// TIA Portal V17 export
// export: Created 2023-12-22T15:05:28.6996043Z, ExportSetting WithDefaults, DisplayName Totally Integrated Automation Portal, DisplayVersion V17, DisplayName TIA Portal Openness, DisplayVersion V17, DisplayName TIA Portal Version Control Interface, DisplayVersion V17, DisplayName STEP 7 Professional, DisplayVersion V17, DisplayName STEP 7 Safety, DisplayVersion V17, DisplayName WinCC Advanced, DisplayVersion V17
FUNCTION_BLOCK "Motors"   // FB240, LAD
{ S7_Optimized_Access := 'FALSE' }
VERSION : 0.1
// stored: AutoNumber false, IsIECCheckEnabled false, SetENOAutomatically false, UDAEnableTagReadback false
   VAR DB_SPECIFIC
      Time_DTL { S7_SetPoint := 'True'} : DTL;
   END_VAR
   VAR_TEMP   // added for the SCL form of the ladder/FBD networks
      _w1 : Bool;
   END_VAR
BEGIN

REGION Network 1: Электролизер / Мешалки
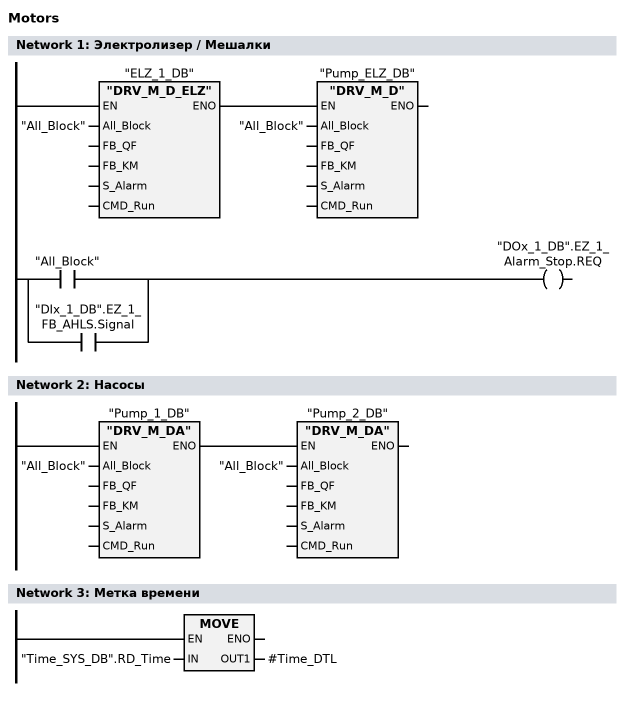
   RUNG wire#powerrail
      "ELZ_1_DB"(All_Block := "All_Block", FB_QF :=, FB_KM :=, S_Alarm :=, CMD_Run :=)
      "Pump_ELZ_DB"(All_Block := "All_Block", FB_QF :=, FB_KM :=, S_Alarm :=, CMD_Run :=)
   END_RUNG
   RUNG wire#powerrail
      Contact( "All_Block" )
      wire#w1
      Coil( "DOx_1_DB".EZ_1_Alarm_Stop.REQ )
   END_RUNG
   RUNG wire#powerrail
      Contact( "DIx_1_DB".EZ_1_FB_AHLS.Signal )
   END_RUNG wire#w1
   // the same network as SCL:
   "ELZ_1_DB"(All_Block := "All_Block", ENO => #_w1);   // "DRV_M_D_ELZ"
   IF #_w1 THEN
       "Pump_ELZ_DB"(All_Block := "All_Block");   // "DRV_M_D"
   END_IF;
   "DOx_1_DB".EZ_1_Alarm_Stop.REQ := "All_Block" OR "DIx_1_DB".EZ_1_FB_AHLS.Signal;
END_REGION

REGION Network 2: Насосы
   RUNG wire#powerrail
      "Pump_1_DB"(All_Block := "All_Block", FB_QF :=, FB_KM :=, S_Alarm :=, CMD_Run :=)
      "Pump_2_DB"(All_Block := "All_Block", FB_QF :=, FB_KM :=, S_Alarm :=, CMD_Run :=)
   END_RUNG
   // the same network as SCL:
   "Pump_1_DB"(All_Block := "All_Block", ENO => #_w1);   // "DRV_M_DA"
   IF #_w1 THEN
       "Pump_2_DB"(All_Block := "All_Block");   // "DRV_M_DA"
   END_IF;
END_REGION

REGION Network 3: Метка времени
   RUNG wire#powerrail
      Move(in := "Time_SYS_DB".RD_Time, out1 => #Time_DTL)
   END_RUNG
   // the same network as SCL:
   #Time_DTL := "Time_SYS_DB".RD_Time;
END_REGION
END_FUNCTION_BLOCK
